(* CODESYS project Übung2.project

Project tree, tasks and I/O mapping:
  CODESYS_Control_Win_V3 : CODESYS Control Win V3, 3S - Smart Software Solutions GmbH, version 3.5.3.60
    application Application
      task Task (cyclic, interval t#20ms, priority 1) calls Blinklicht
      program Blinklicht [ST]
      function block blink [ST]
*)

// CODESYS_Control_Win_V3/Application/Blinklicht
PROGRAM Blinklicht
VAR 
	feld AT %QX10.0: ARRAY[1..8] OF BOOL; 
	(* 8 Signale ab %QX10.0 *) 
	auf: R_TRIG; 
	takt: blink;(*FB der nach Ablauf der Brenndauer*) 
	(* eine steigende Flanke liefert*) 
	i: INT := 1; (* wird mit 1 initial. *) 
END_VAR

END_PROGRAM

// CODESYS_Control_Win_V3/Application/blink
FUNCTION_BLOCK blink 
VAR_INPUT 
	enable: BOOL; 
	thigh, 
	tlow: TIME; 
END_VAR 
VAR_OUTPUT 
	Q: BOOL; (*Blinksignal*) 
END_VAR 
VAR 
	an, aus: TP; (* Timerbaustein für Impulszeit *) 
END_VAR

	an (IN := ENABLE & NOT aus.Q, 
	PT:= thigh); 
	aus(IN := NOT an.Q, PT := tlow); 
	Q := an.Q; 
END_FUNCTION_BLOCK

END_FUNCTION_BLOCK
